PROGRAM MAIN
VAR
END_VAR

POU_SM01_LineBend();

POU_SA01_ReadScanners();

POU_DT01_EnableDriveTrain();
POU_DT02_MotorControl();

END_PROGRAM

(* stored: Version 1.1.0.1, ProductVersion 3.1.4022.7
   POU MAIN: Id {412e421b-8a23-4559-9dfe-993367fdf278}, SpecialFunc None *)
